FUNCTION_BLOCK irrigation_Main_Controller
VAR_INPUT
	Moisture : bool;
	T_Max : time;
END_VAR

VAR_IN_OUT
	State : irrigation_State;
END_VAR

VAR
	man_mode : bool;
	timeout : bool;
	run_valve : bool;
	TON0 : TON;
	TOF0 : TOF;
END_VAR

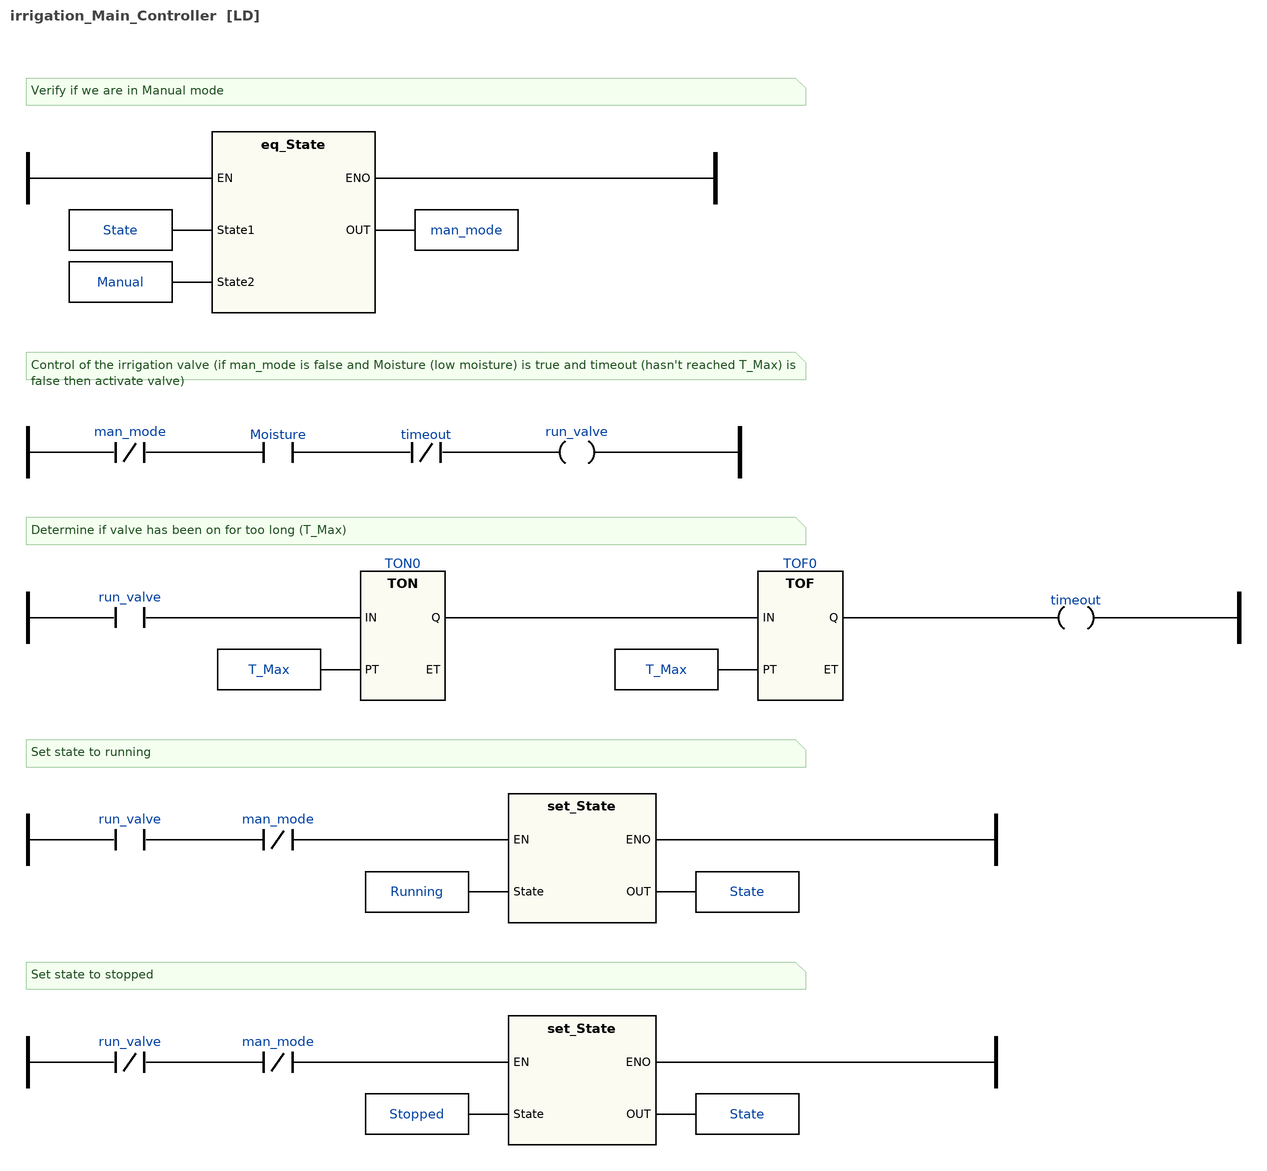
(* LD diagram, written out as Structured Text *)
(* Verify if we are in Manual mode *)
man_mode := eq_State(State, Manual);
(* Control of the irrigation valve (if man_mode is false and Moisture (low moisture) is true and timeout (hasn't reached T_Max) is false then activate valve) *)
run_valve := NOT man_mode AND Moisture AND NOT timeout;
(* Determine if valve has been on for too long (T_Max) *)
TON0(IN := run_valve, PT := T_Max);
TOF0(IN := TON0.Q, PT := T_Max);
timeout := TOF0.Q;
(* Set state to running *)
IF run_valve AND NOT man_mode THEN State := set_State(Running); END_IF;
(* Set state to stopped *)
IF NOT run_valve AND NOT man_mode THEN State := set_State(Stopped); END_IF;
END_FUNCTION_BLOCK
